PROGRAM prgIO
VAR;
END_VAR

// ~~~~~ CoE I/O ~~~~~
(*
PLC Inputs

0x2191:01 (bit 0) Probe 1 signal
0x2199:01 Probe 1 positive latched
0x219A:01 Probe 1 negative latched

PLC Outputs

0x20AA:01 Probing cycle command
0x2195:01 Probe 1 enable
*)

// Scan Toggle
gvlServo.bExecute := NOT gvlServo.bExecute;

// ~ Inputs ~
// Probe 1 Signal : 2191:01
gvlServo.coeRead(Axis:= gvlServo.servo1Interface.ioAxisRef,
				  Index := 16#2191,
				  SubIndex := 16#01,
				  Execute := gvlServo.bExecute,
				  Busy =>,
				  pDstBuf := ADR(gvlIO.stInputs.coeProbe1Signal),
				  BufLen := SIZEOF(gvlIO.stInputs.coeProbe1Signal));

// Probe 1 Positive Latched: 2199:01
gvlServo.coeRead(Axis:= gvlServo.servo1Interface.ioAxisRef,
				  Index := 16#2199,
				  SubIndex := 16#01,
				  Execute := gvlServo.bExecute,
				  Busy =>,
				  pDstBuf := ADR(gvlIO.stInputs.coeProbe1PosLatch),
				  BufLen := SIZEOF(gvlIO.stInputs.coeProbe1PosLatch));

// Probe 1 Negative Latched: 219A:01
gvlServo.coeRead(Axis:= gvlServo.servo1Interface.ioAxisRef,
				  Index := 16#219A,
				  SubIndex := 16#01,
				  Execute := gvlServo.bExecute,
				  Busy =>,
				  pDstBuf := ADR(gvlIO.stInputs.coeProbe1NegLatch),
				  BufLen := SIZEOF(gvlIO.stInputs.coeProbe1NegLatch));

// ~ Outputs ~
// Probing Cycle Command : 20AA:01
	gvlServo.coeWrite(
		Axis:= gvlServo.servo1Interface.ioAxisRef, 
		Index:= 16#20AA, 
		SubIndex:= 16#01, 
		pSrcBuf:= ADR(gvlIO.stOutputs.coeProbingCycleCommand), 
		BufLen:= SIZEOF(gvlIO.stOutputs.coeProbingCycleCommand), 
		Execute:= gvlServo.bExecute);
// Probe 1 Enable : 2195:01
	gvlServo.coeWrite(
		Axis:= gvlServo.servo1Interface.ioAxisRef, 
		Index:= 16#2195, 
		SubIndex:= 16#01, 
		pSrcBuf:= ADR(gvlIO.stOutputs.coeProbe1Enable), 
		BufLen:= SIZEOF(gvlIO.stOutputs.coeProbingCycleCommand), 
		Execute:= gvlServo.bExecute);

END_PROGRAM

(* stored: Version 1.1.0.1, ProductVersion 3.1.4024.12
   POU prgIO: Id {8caf3471-a93f-413d-a856-c301020de24e}, SpecialFunc None *)
